FUNCTION_BLOCK Skill_Position_anfahren_erweitert	IMPLEMENTS I_Skill_RoboterErweitert
VAR_INPUT
	// Zu verwendetes Objekt
	Objekt						:I_Objekt_Roboter;	
	
	sMessdaten					:Kraftvariablen; 
	
	// Betriebsvariablen
	eSysCommand					:eSystemCommand; 						// Systembefehl an Skill
	eSysState					:eSystemState;							// Momentaner Zustand des Systems
	
END_VAR
VAR_OUTPUT
	iErrorID					:INT;									// Fehlercode für System
END_VAR
VAR
	// Managementvariablen
	iState				:eSkillState;									// Information über Zustand von Skill
	bGestartet			:BOOL;
	bGestoppt			:BOOL;
	
	// Zustandsvariablen
	bStarten			:BOOL;
	bStoppen			:BOOL;
	bObjektFertig		:BOOL;
	bErreicht			:BOOL;				
	bLimit				:BOOL;				
	bSkillFertig		:BOOL;
	bFehler				:BOOL;
	bResetten			:BOOL;
	
	// Prozessparameter
	eRoboterPos		 			:sRoboterProzessVariablen;
	sLimit						:sKraftVariablen;
	sErreicht					:sKraftVariablen;
	
END_VAR

// Fehlerüberwachung
IF bFehler THEN
	iState := 3;
END_IF

//_______________________________________________________________
// Reaktion auf Input-Variablen:
	// Stoppen
	IF eSysCommand = 3 THEN
		bStoppen := M_Stop();
	ELSE 
		bStoppen := FALSE;
	END_IF

	// Resetten 
	IF eSysCommand = 4 THEN
		bResetten := M_Reset();
	ELSE
		bResetten := FALSE;
	END_IF
//_______________________________________________________________
// Zustandsmanagement
CASE iState OF 
0: 	// BEREIT	
		// DO
		IF Objekt.P_State = 3 THEN		// Objekt wurde eingeschalten
			bStarten := TRUE;
		END_IF
		
		// TRANSITION
		IF bStarten	 THEN		
			bStarten := FALSE;
			iState := 1;	
		END_IF
		
		
// _________________________________________________________________________________________________________________________
1: 	// LAUFEND
		// DO		
			// Auswerten
			M_Auswertung();
				
			// Stoppen durch Sysezm
			IF bStoppen THEN																								// Transition wenn System das Orbjekt stoppt
				bGestoppt := TRUE;
			END_IF
			
			// Objekt hat sich selber gestoppt
			IF Objekt.P_State = 4 THEN																							// Objekt hat Prozess abgeschlossen
				bObjektFertig := TRUE;																							// Objekt ist fertig und wieder bereit
			END_IF
			
			// Limit Erreicht -> Objekt wird gestoppt
			IF bLimit THEN
				Objekt.M_Stop();
			END_IF
			
			// Wert Erreicht -> Objekt wird gestoppt
			IF bErreicht THEN
				Objekt.M_Stop();
			END_IF
			
		// TRANSITION 
		IF bGestoppt THEN																								// Transition zu BEREIT
			bGestoppt := FALSE;													
			iState := 0;
		END_IF
		
		IF bObjektFertig THEN																							// Transition zu ABGESCHLOSSEN
			bObjektFertig := FALSE;																							// Skill wird nicht mehr ausgeführt
			iState := 2;																									// Objekt ist fertig und wieder bereit
		END_IF
		
		IF bLimit AND Objekt.P_State = 5 THEN																							// Transition zu LIMIT
			bLimit := FALSE;
			iState := 4;
		END_IF
		
		IF bErreicht AND Objekt.P_State = 5 THEN																							// Transition zu ERREICHT
			bErreicht := FALSE;
			iState := 5;
		END_IF
			
// _________________________________________________________________________________________________________________________			
2: 	// ABGESCHLOSSEN
		// DO
		IF Objekt.P_State = 1 THEN																							// Objekt wurde geresettet
			bSkillFertig := TRUE;									
		END_IF
			
		//  TRANSITION
		IF bSkillFertig THEN
			bSkillFertig := FALSE;																																											// Resetten von Objekt
			iState := 0;
		END_IF
		
// _________________________________________________________________________________________________________________________
3: 	// FEHLER
		// DO 	
		
		// TRANSITION
		IF bResetten THEN
			iState := 0;
		END_IF
		
// _________________________________________________________________________________________________________________________			
4: 	// LIMIT
		// DO		
		M_Reset();
		
		IF Objekt.P_State = 1 THEN																								// Objekt wurde geresettet
			bResetten := TRUE;								
		END_IF
	
		// TRANSITION
		IF bResetten THEN
			bResetten := FALSE;
			iState := 0;
		END_IF
			
// _________________________________________________________________________________________________________________________
5: 	// ERREICHT		
		// DO 
		M_Reset();
		
		IF Objekt.P_State = 1 THEN																							// Objekt wurde geresettet
			bSkillFertig := TRUE;									
		END_IF
		
		// TRANSITION
		IF bSkillFertig THEN
			bSkillFertig := FALSE;
			iState := 0;
		END_IF
		
END_CASE

METHOD M_Auswertung : BOOL
VAR_INPUT
END_VAR
VAR
	bLimit_x		:BOOL;
	bLimit_y		:BOOL;
	bLimit_z		:BOOL;
	
	bErreicht_x		:BOOL;
	bErreicht_y		:BOOL;
	bErreicht_z		:BOOL;
END_VAR
IF sLimit.Fx <> 0 THEN
	IF ABS(sMessdaten.Fx) >= ABS(sLimit.Fx) THEN
		bLimit_x := TRUE;
	END_IF
END_IF

IF sLimit.Fy <> 0 THEN
	IF ABS(sMessdaten.Fy) >= ABS(sLimit.Fy) THEN
		bLimit_y := TRUE;
	END_IF
END_IF

IF sLimit.Fz <> 0 THEN
	IF ABS(sMessdaten.Fz) >= ABS(sLimit.Fz) THEN
		bLimit_x := TRUE;
	END_IF
END_IF

// Auswertung von Erreicht-Wert
IF sErreicht.Fx <> 0 THEN
	IF ABS(sMessdaten.Fx) >= ABS(sErreicht.Fx) THEN
		bErreicht_x := TRUE;
	END_IF
END_IF

IF sErreicht.Fy <> 0 THEN
	IF ABS(sMessdaten.Fy) >= ABS(sErreicht.Fy) THEN
		bErreicht_y := TRUE;
	END_IF
END_IF

IF sErreicht.Fz <> 0 THEN
	IF ABS(sMessdaten.Fz) >= ABS(sErreicht.Fz) THEN
		bErreicht_z := TRUE;
	END_IF
END_IF

IF bLimit_x OR bLimit_y OR bLimit_z THEN
	bLimit := TRUE;
END_IF

IF bErreicht_x OR bErreicht_y OR bErreicht_z THEN
	bErreicht := TRUE;
END_IF
END_METHOD

METHOD M_Reset : BOOL
Objekt.M_Reset();
END_METHOD

METHOD M_Start : BOOL
// Prüfen von Bedingungen
	// Ist das  System im korrekten Status
	IF eSysState = 1 OR eSysState = 2 THEN
		// Ist der Skill im korrekten Status 
		IF iState = 0 THEN
			// Prüfen auf Fehler (Muss ergänzt werden)
			
				Objekt.P_Prozessparameter := eRoboterPos;
				Objekt.M_Start();	
		END_IF
	END_IF
END_METHOD

METHOD M_Stop : BOOL
Objekt.M_Stop();
END_METHOD

PROPERTY P_Erreicht : sKraftVariablen
SET
sErreicht := P_Erreicht;
END_SET
END_PROPERTY

PROPERTY P_Limit : sKraftVariablen
SET
sLimit := P_Limit;
END_SET
END_PROPERTY

PROPERTY P_RobotParam : sRoboterProzessVariablen
SET
eRoboterPos := P_RobotParam;
END_SET
END_PROPERTY

PROPERTY P_State : eSkillState
GET
P_State := iState;
END_GET
END_PROPERTY

END_FUNCTION_BLOCK

(* stored: Version 1.1.0.1
   POU Skill_Position_anfahren_erweitert: Id {20d2290a-8794-4965-a133-9ad0acf7b5f9}, SpecialFunc None
   Folder 01_Steuerungsmethoden: Id {24108a3b-139b-4abc-9ee1-f7b20236da36}
   Folder 02_Steuerungseigenschaften: Id {81dfad2e-6b4f-4546-926f-b569be2ebe07}
   Folder 03_Prozessmethoden: Id {2f427658-d188-4219-be86-1c49d4b928f8}
   Folder 04_Prozesseigenschaften: Id {a2461b16-3250-454b-89ff-eb78ad4ff0ad}
   Method M_Auswertung: Id {466dc7d6-1b9c-4401-885b-20f06b59f3fc}
   Method M_Reset: Id {2e9015dd-f485-4671-90bc-8e693338c9f5}
   Method M_Start: Id {bcb53f09-8eee-41d0-920b-9b5bddfe5634}
   Method M_Stop: Id {ec311155-7585-4e1e-a8e1-ec23ba2ba7f7}
   Property P_Erreicht: Id {65ff26fd-bd5b-4448-b176-bea996d64888}
   Set Set: Id {e9f2cea9-274a-4473-a8e1-84efb25603cf}
   Property P_Limit: Id {d6272a96-2f33-45dc-be76-82f80d521d23}
   Set Set: Id {997dbb89-0df6-40fe-8bb6-a14113d7e3ed}
   Property P_RobotParam: Id {8624615e-7d1d-4a98-af5b-70ce2c99259c}
   Set Set: Id {d4382561-34b8-4238-9b23-e9a998a335f2}
   Property P_State: Id {a7d51d8e-fee2-4f41-ac35-d1a2b9f3cc03}
   Get Get: Id {a4e9133e-8c8c-4005-84ab-77b9f037aa9d} *)
